(* IEC 61131-3 sources: verifaps-lib/share/PPU.stold (part 13) *)

(* ---- Scenario8_Final.xml.st ---- *)
TYPE
    Magazin_states_t : (Green_Lamp , Init , Interstep , Magazin_Init , Magazin_Init_2 , Slider_Move_Back , Start_Magazin , Step0 , Step1 , convey);
    Stamp_states_t : (Green_Lamp , Init , Interstep , Interstep_2 , StampProcess , StampSliderBack , StampSliderForward , Stamp_Init_1 , Stamp_Init_2 , Stamp_Init_3 , Stamp_Init_4 , Start_Stamp , Step0 , Step1 , Step2);
    Crane_states_t : (Crane_Go_Up , Crane_Go_Up_White , Crane_Init , Crane_Init_2 , Crane_Lift_At_Stamp , Crane_Lift_At_Stamp2 , Crane_Lift_Conveyor , Crane_Lift_Conveyor2 , Crane_Lift_Conveyor_Black , Crane_Lift_Magazin , Crane_Lift_Magazin_Metallic , Crane_Lift_Magazine_White , Crane_Lift_NOT_Metallic_Black , Crane_Lower , Crane_On_Conveyor , Crane_On_Conveyor_Metallic , Crane_On_Conveyor_Metallic2 , Crane_On_Conveyor_Not_Metallica_Black , Crane_On_Stamp_Metallic , Crane_On_Stamp_Metallic2 , Crane_On_Stamp_Metallic2_Lower , Crane_On_Stamp_Stop_Black , Crane_On_Stamp_White , Crane_Turn_Left_Back_To_Stamp , Crane_Turn_Left_From_Stamp , Crane_Turn_Left_Metallic , Crane_Turn_Left_Metallic2 , Crane_Turn_Left_NOT_Metallic , Crane_Turn_Left_NOT_Metallic_Black , Crane_Turn_Left_White , Crane_Turn_Right_From_Stamp , Init , Interstep , Interstep_2 , Interstep_3 , Interstep_4 , Lower_Crane , Magazin_Stop , Magazin_Stop_Black , Magazin_Stop_Final , No_Workpiece_ready , Reset_interconnect , Stamp_Pressure_Profile_Set_Metallic , Stamp_Pressure_Profile_Set_White , Start_Crane , Step0 , Step2 , Step3 , Step4 , Suck_At_Stamp , Suck_At_Stamp2 , TimeDelay , Turn_Right , Turn_Right_Black , Turn_Right_Final , pause , release , release2 , release_Black , release_Workpiece , release_Workpiece_White);
END_TYPE

FUNCTION_BLOCK Magazin
    VAR_INPUT  CraneDown : BOOL; END_VAR {*Irwxp*}
    VAR_OUTPUT  CraneLower : BOOL; END_VAR {*Orwxp*}
    VAR_INPUT  CraneOnConveyor : BOOL; END_VAR {*Irwxp*}
    VAR_INPUT  CraneOnMagazin : BOOL; END_VAR {*Irwxp*}
    VAR_INPUT  CraneSucked : BOOL; END_VAR {*Irwxp*}
    VAR_OUTPUT  CraneTurnClockwise : BOOL; END_VAR {*Orwxp*}
    VAR_OUTPUT  CraneTurnCounterclockwise : BOOL; END_VAR {*Orwxp*}
    VAR_INPUT  CraneUp : BOOL; END_VAR {*Irwxp*}
    VAR_OUTPUT  MagazinGreenLamp : BOOL; END_VAR {*Orwxp*}
    VAR_OUTPUT  MagazinSlider : BOOL; END_VAR {*Orwxp*}
    VAR_OUTPUT  MagazinVacuumOff : BOOL; END_VAR {*Orwxp*}
    VAR_OUTPUT  MagazinVacuumOn : BOOL; END_VAR {*Orwxp*}
    VAR_OUTPUT  MagazinWhiteLamp : BOOL; END_VAR {*Orwxp*}
    VAR  SFCInit : BOOL; END_VAR {*Lrwxp*}
    VAR_INPUT  SFCReset : BOOL; END_VAR {*Irwxp*}
    VAR_INPUT  SliderMovedOut : BOOL; END_VAR {*Irwxp*}
    VAR_INPUT  SliderNotMovedOut : BOOL; END_VAR {*Irwxp*}
    VAR_INPUT  StartButtonMagazin : BOOL; END_VAR {*Irwxp*}
    VAR_OUTPUT  StartCommandMagazin : BOOL; END_VAR {*Orwxp*}
    VAR_INPUT  StartVar : BOOL; END_VAR {*Irwxp*}
    VAR_INPUT  WorkpieceReady : BOOL; END_VAR {*Irwxp*}
    VAR  _state : Magazin_states_t; END_VAR {*Lrwxp*}
    VAR  _transit : BOOL; END_VAR {*Lrwxp*}
    VAR  interconnectMagazinStartCommand : BOOL; END_VAR {*Lrwxp*}

    CASE _state OF
        Magazin_states_t#Green_Lamp:
            _transit := FALSE;
            MagazinGreenLamp := TRUE;
            interconnectMagazinStartCommand := FALSE;
            IF TRUE THEN
                _transit := TRUE;
                _state := Magazin_states_t#Magazin_Init;
            END_IF;

        Magazin_states_t#Init:
            _transit := FALSE;
            IF TRUE THEN
                _transit := TRUE;
                _state := Magazin_states_t#Start_Magazin;
            END_IF;

        Magazin_states_t#Interstep:
            _transit := FALSE;
            StartCommandMagazin := TRUE;
            IF StartVar THEN
                _transit := TRUE;
                _state := Magazin_states_t#convey;
            END_IF;

        Magazin_states_t#Magazin_Init:
            _transit := FALSE;
            MagazinSlider := TRUE;
            IF TRUE THEN
                _transit := TRUE;
                _state := Magazin_states_t#Magazin_Init_2;
            END_IF;

        Magazin_states_t#Magazin_Init_2:
            _transit := FALSE;
            MagazinSlider := FALSE;
            IF TRUE THEN
                _transit := TRUE;
                _state := Magazin_states_t#Interstep;
            END_IF;

        Magazin_states_t#Slider_Move_Back:
            _transit := FALSE;
            IF ((SliderMovedOut = TRUE) AND (SliderNotMovedOut = FALSE)) THEN
                MagazinSlider := FALSE;
            END_IF;
            IF CraneUp THEN
                _transit := TRUE;
                _state := Magazin_states_t#Step1;
            END_IF;

        Magazin_states_t#Start_Magazin:
            _transit := FALSE;
            MagazinSlider := FALSE;
            MagazinGreenLamp := FALSE;
            StartVar := FALSE;
            StartCommandMagazin := FALSE;
            IF (StartButtonMagazin = TRUE) THEN
                interconnectMagazinStartCommand := TRUE;
            END_IF;
            IF interconnectMagazinStartCommand THEN
                _transit := TRUE;
                _state := Magazin_states_t#Green_Lamp;
            END_IF;

        Magazin_states_t#Step0:
            _transit := FALSE;
            IF CraneDown THEN
                _transit := TRUE;
                _state := Magazin_states_t#Slider_Move_Back;
            END_IF;

        Magazin_states_t#Step1:
            _transit := FALSE;
            IF CraneOnConveyor THEN
                _transit := TRUE;
                _state := Magazin_states_t#Interstep;
            END_IF;

        Magazin_states_t#convey:
            _transit := FALSE;
            IF SliderNotMovedOut THEN
                MagazinSlider := TRUE;
            END_IF;
            IF CraneOnMagazin THEN
                _transit := TRUE;
                _state := Magazin_states_t#Step0;
            END_IF;

            END_CASE;
END_FUNCTION_BLOCK

PROGRAM Main

VAR  Actuator_AnalogCranePressure : INT; END_VAR {*Lrwxp*}
VAR  Actuator_CraneLower : BOOL; END_VAR {*Lrwxp*}
VAR  Actuator_CraneTurnClockwise : BOOL; END_VAR {*Lrwxp*}
VAR  Actuator_CraneTurnCounterclockwise : BOOL; END_VAR {*Lrwxp*}
VAR  Actuator_MagazinGreenLamp : BOOL; END_VAR {*Lrwxp*}
VAR  Actuator_MagazinSlider : BOOL; END_VAR {*Lrwxp*}
VAR  Actuator_MagazinVacuumOff : BOOL; END_VAR {*Lrwxp*}
VAR  Actuator_MagazinVacuumOn : BOOL; END_VAR {*Lrwxp*}
VAR  Actuator_MagazinWhiteLamp : BOOL; END_VAR {*Lrwxp*}
VAR  Actuator_StampGreenLamp : BOOL; END_VAR {*Lrwxp*}
VAR  Actuator_StampPusher : BOOL; END_VAR {*Lrwxp*}
VAR  Actuator_StampSliderMovedIn : BOOL; END_VAR {*Lrwxp*}
VAR  Actuator_StampSliderMovedOut : BOOL; END_VAR {*Lrwxp*}
VAR  Actuator_StampWhiteLamp : BOOL; END_VAR {*Lrwxp*}
VAR  Crane : Crane; END_VAR {*Lrwxp*}
VAR  Mag : Magazin; END_VAR {*Lrwxp*}
VAR  Sensor_CraneDown : BOOL; END_VAR {*Lrwxp*}
VAR  Sensor_CraneOnConveyor : BOOL; END_VAR {*Lrwxp*}
VAR  Sensor_CraneOnMagazin : BOOL; END_VAR {*Lrwxp*}
VAR  Sensor_CranePosition : BOOL; END_VAR {*Lrwxp*}
VAR  Sensor_CranePositionStamp : BOOL; END_VAR {*Lrwxp*}
VAR  Sensor_CraneSucked : BOOL; END_VAR {*Lrwxp*}
VAR  Sensor_CraneUp : BOOL; END_VAR {*Lrwxp*}
VAR  Sensor_MagazinCapacitiveSensor : BOOL; END_VAR {*Lrwxp*}
VAR  Sensor_MagazinEmergencyStop : BOOL; END_VAR {*Lrwxp*}
VAR  Sensor_MagazinOpticalSensor : BOOL; END_VAR {*Lrwxp*}
VAR  Sensor_MagazinSwitchManuellAutomatic : BOOL; END_VAR {*Lrwxp*}
VAR  Sensor_SliderMovedOut : BOOL; END_VAR {*Lrwxp*}
VAR  Sensor_SliderNotMovedOut : BOOL; END_VAR {*Lrwxp*}
VAR  Sensor_StampEmergencyStop : BOOL; END_VAR {*Lrwxp*}
VAR  Sensor_StampLowered : BOOL; END_VAR {*Lrwxp*}
VAR  Sensor_StampSliderFilled : BOOL; END_VAR {*Lrwxp*}
VAR  Sensor_StampSliderSensorMovedIn : BOOL; END_VAR {*Lrwxp*}
VAR  Sensor_StampSliderSensorMovedOut : BOOL; END_VAR {*Lrwxp*}
VAR  Sensor_StampStartButton : BOOL; END_VAR {*Lrwxp*}
VAR  Sensor_StampSwitchManuellAutomatic : BOOL; END_VAR {*Lrwxp*}
VAR  Sensor_StampUp : BOOL; END_VAR {*Lrwxp*}
VAR  Sensor_StartButtonMagazin : BOOL; END_VAR {*Lrwxp*}
VAR  Sensor_WorkpieceReady : BOOL; END_VAR {*Lrwxp*}
VAR  Stamp : Stamp; END_VAR {*Lrwxp*}
Mag.SliderNotMovedOut := Sensor_SliderNotMovedOut;
Mag.SliderMovedOut := Sensor_SliderMovedOut;
Mag.CraneOnMagazin := Sensor_CraneOnMagazin;
Mag.CraneDown := Sensor_CraneDown;
Mag.CraneUp := Sensor_CraneUp;
Mag.CraneOnConveyor := Sensor_CraneOnConveyor;
Mag.WorkpieceReady := Sensor_WorkpieceReady;
Mag.StartButtonMagazin := Sensor_StartButtonMagazin;
Actuator_MagazinSlider := Mag.MagazinSlider;
Actuator_MagazinGreenLamp := Mag.MagazinGreenLamp;
Crane.CraneUp := Sensor_CraneUp;
Crane.CraneOnConveyor := Sensor_CraneOnConveyor;
Crane.CraneDown := Sensor_CraneDown;
Crane.CraneSucked := Sensor_CraneSucked;
Crane.CraneOnMagazin := Sensor_CraneOnMagazin;
Crane.MagazinCapacitiveSensor := Sensor_MagazinCapacitiveSensor;
Crane.CranePositionStamp := Sensor_CranePositionStamp;
Crane.SliderMovedOut := Sensor_SliderMovedOut;
Crane.WorkpieceReady := Sensor_WorkpieceReady;
Crane.MagazinOpticalSensor := Sensor_MagazinOpticalSensor;
Crane.StampSliderFilled := Sensor_StampSliderFilled;
Crane.StampSliderSensorMovedOut := Sensor_StampSliderSensorMovedOut;
Crane.StampLowered := Sensor_StampLowered;
Crane.StartButtonMagazin := Sensor_StartButtonMagazin;
Actuator_CraneTurnCounterclockwise := Crane.CraneTurnCounterclockwise;
Actuator_CraneTurnClockwise := Crane.CraneTurnClockwise;
Actuator_CraneLower := Crane.CraneLower;
Actuator_MagazinVacuumOff := Crane.MagazinVacuumOff;
Actuator_MagazinVacuumOn := Crane.MagazinVacuumOn;
Actuator_AnalogCranePressure := Crane.AnalogCranePressure;
Stamp.StampSliderSensorMovedOut := Sensor_StampSliderSensorMovedOut;
Stamp.StampSliderSensorMovedIn := Sensor_StampSliderSensorMovedIn;
Stamp.StampSliderFilled := Sensor_StampSliderFilled;
Stamp.StampUp := Sensor_StampUp;
Stamp.StampLowered := Sensor_StampLowered;
Stamp.CraneDown := Sensor_CraneDown;
Stamp.CraneUp := Sensor_CraneUp;
Stamp.CraneSucked := Sensor_CraneSucked;
Stamp.CranePositionStamp := Sensor_CranePositionStamp;
Stamp.CraneOnConveyor := Sensor_CraneOnConveyor;
Stamp.StampStartButton := Sensor_StampStartButton;
Actuator_StampSliderMovedOut := Stamp.StampSliderMovedOut;
Actuator_StampSliderMovedIn := Stamp.StampSliderMovedIn;
Actuator_StampWhiteLamp := Stamp.StampWhiteLamp;
Actuator_StampPusher := Stamp.StampPusher;
Actuator_StampGreenLamp := Stamp.StampGreenLamp;
IF (Sensor_StampEmergencyStop AND Sensor_MagazinEmergencyStop) THEN
    Mag();
    Crane();
    Stamp();
    IF (Actuator_MagazinGreenLamp AND Actuator_StampGreenLamp) THEN
        IF ((Stamp.StartCommandStamp AND Crane.StartCommandCrane) AND Mag.StartCommandMagazin) THEN
            Crane.StartVar := TRUE;
            Mag.StartVar := TRUE;
            Stamp.StartVar := TRUE;
        END_IF;
    END_IF;
    Crane.SFCReset := FALSE;
    Mag.SFCReset := FALSE;
    Stamp.SFCReset := FALSE;
ELSEIF (NOT Sensor_StampEmergencyStop OR NOT Sensor_MagazinEmergencyStop) THEN
    Actuator_MagazinSlider := FALSE;
    Actuator_CraneLower := FALSE;
    Actuator_MagazinVacuumOn := FALSE;
    Actuator_MagazinVacuumOff := TRUE;
    Actuator_MagazinGreenLamp := FALSE;
    Actuator_CraneTurnCounterclockwise := FALSE;
    Actuator_CraneTurnClockwise := FALSE;
    Actuator_StampSliderMovedOut := TRUE;
    Actuator_StampSliderMovedIn := FALSE;
    Actuator_StampGreenLamp := FALSE;
    Actuator_StampPusher := FALSE;
    Actuator_AnalogCranePressure := INT#0;
    Crane.SFCReset := TRUE;
    Mag.SFCReset := TRUE;
    Stamp.SFCReset := TRUE;
    Crane.StartVar := FALSE;
    Mag.StartVar := FALSE;
    Stamp.StartVar := FALSE;
END_IF;
END_PROGRAM
FUNCTION_BLOCK Stamp
VAR_INPUT  CraneDown : BOOL; END_VAR {*Irwxp*}
VAR_INPUT  CraneOnConveyor : BOOL; END_VAR {*Irwxp*}
VAR_INPUT  CranePositionStamp : BOOL; END_VAR {*Irwxp*}
VAR_INPUT  CraneSucked : BOOL; END_VAR {*Irwxp*}
VAR_INPUT  CraneUp : BOOL; END_VAR {*Irwxp*}
VAR  Duration : TIME := TIME#500.0ms; END_VAR {*Lrwxp*}
VAR  SFCInit : BOOL; END_VAR {*Lrwxp*}
VAR_INPUT  SFCReset : BOOL; END_VAR {*Irwxp*}
VAR_OUTPUT  StampGreenLamp : BOOL; END_VAR {*Orwxp*}
VAR_INPUT  StampLowered : BOOL; END_VAR {*Irwxp*}
VAR_OUTPUT  StampPressure : BOOL; END_VAR {*Orwxp*}
VAR_OUTPUT  StampPusher : BOOL; END_VAR {*Orwxp*}
VAR_INPUT  StampSliderFilled : BOOL; END_VAR {*Irwxp*}
VAR_OUTPUT  StampSliderMovedIn : BOOL; END_VAR {*Orwxp*}
VAR_OUTPUT  StampSliderMovedOut : BOOL; END_VAR {*Orwxp*}
VAR_INPUT  StampSliderSensorMovedIn : BOOL; END_VAR {*Irwxp*}
VAR_INPUT  StampSliderSensorMovedOut : BOOL; END_VAR {*Irwxp*}
VAR_INPUT  StampStartButton : BOOL; END_VAR {*Irwxp*}
VAR_INPUT  StampUp : BOOL; END_VAR {*Irwxp*}
VAR_OUTPUT  StampWhiteLamp : BOOL; END_VAR {*Orwxp*}
VAR_OUTPUT  StartCommandStamp : BOOL; END_VAR {*Orwxp*}
VAR_INPUT  StartVar : BOOL; END_VAR {*Irwxp*}
VAR  Timer : TON; END_VAR {*Lrwxp*}
VAR  _state : Stamp_states_t; END_VAR {*Lrwxp*}
VAR  _transit : BOOL; END_VAR {*Lrwxp*}
VAR  interconnect : BOOL; END_VAR {*Lrwxp*}
VAR  interconnectStampStartCommand : BOOL; END_VAR {*Lrwxp*}

CASE _state OF
    Stamp_states_t#Green_Lamp:
        _transit := FALSE;
        StampGreenLamp := TRUE;
        interconnectStampStartCommand := FALSE;
        IF TRUE THEN
            _transit := TRUE;
            _state := Stamp_states_t#Stamp_Init_1;
        END_IF;

    Stamp_states_t#Init:
        _transit := FALSE;
        IF TRUE THEN
            _transit := TRUE;
            _state := Stamp_states_t#Start_Stamp;
        END_IF;

    Stamp_states_t#Interstep:
        _transit := FALSE;
        StartCommandStamp := TRUE;
        IF StartVar THEN
            _transit := TRUE;
            _state := Stamp_states_t#Interstep_2;
        END_IF;

    Stamp_states_t#Interstep_2:
        _transit := FALSE;
        IF StampSliderFilled THEN
            _transit := TRUE;
            _state := Stamp_states_t#Step0;
        END_IF;

    Stamp_states_t#StampProcess:
        _transit := FALSE;
        StampSliderMovedIn := FALSE;
        StampPusher := TRUE;
        IF StampLowered THEN
            _transit := TRUE;
            _state := Stamp_states_t#Step1;
        END_IF;

    Stamp_states_t#StampSliderBack:
        _transit := FALSE;
        StampSliderMovedIn := TRUE;
        StampSliderMovedOut := FALSE;
        IF StampSliderSensorMovedIn THEN
            _transit := TRUE;
            _state := Stamp_states_t#StampProcess;
        END_IF;

    Stamp_states_t#StampSliderForward:
        _transit := FALSE;
        StampPusher := FALSE;
        StampSliderMovedOut := TRUE;
        IF ((StampLowered = FALSE) AND (StampUp = TRUE)) THEN
            interconnect := FALSE;
        END_IF;
        Timer(IN := FALSE, PT := TIME#1.0ms);
        IF StampSliderMovedOut THEN
            _transit := TRUE;
            _state := Stamp_states_t#Step2;
        END_IF;

    Stamp_states_t#Stamp_Init_1:
        _transit := FALSE;
        StampSliderMovedIn := TRUE;
        StampSliderMovedOut := FALSE;
        IF StampSliderSensorMovedIn THEN
            _transit := TRUE;
            _state := Stamp_states_t#Stamp_Init_2;
        END_IF;

    Stamp_states_t#Stamp_Init_2:
        _transit := FALSE;
        StampSliderMovedIn := FALSE;
        StampSliderMovedOut := TRUE;
        IF StampSliderSensorMovedOut THEN
            _transit := TRUE;
            _state := Stamp_states_t#Stamp_Init_3;
        END_IF;

    Stamp_states_t#Stamp_Init_3:
        _transit := FALSE;
        StampPusher := TRUE;
        IF StampLowered THEN
            _transit := TRUE;
            _state := Stamp_states_t#Stamp_Init_4;
        END_IF;

    Stamp_states_t#Stamp_Init_4:
        _transit := FALSE;
        StampPusher := FALSE;
        IF StampUp THEN
            _transit := TRUE;
            _state := Stamp_states_t#Interstep;
        END_IF;

    Stamp_states_t#Start_Stamp:
        _transit := FALSE;
        StampSliderMovedOut := FALSE;
        StampSliderMovedIn := FALSE;
        StampPusher := FALSE;
        StampGreenLamp := FALSE;
        StampPressure := FALSE;
        StartCommandStamp := FALSE;
        IF (StampStartButton = TRUE) THEN
            interconnectStampStartCommand := TRUE;
        END_IF;
        IF interconnectStampStartCommand THEN
            _transit := TRUE;
            _state := Stamp_states_t#Green_Lamp;
        END_IF;

    Stamp_states_t#Step0:
        _transit := FALSE;
        IF CraneUp THEN
            _transit := TRUE;
            _state := Stamp_states_t#StampSliderBack;
        END_IF;

    Stamp_states_t#Step1:
        _transit := FALSE;
        Timer(IN := StampLowered, PT := TIME#);
        interconnect := Timer.Q;
        IF interconnect THEN
            _transit := TRUE;
            _state := Stamp_states_t#StampSliderForward;
        END_IF;

    Stamp_states_t#Step2:
        _transit := FALSE;
        IF (CraneOnConveyor AND NOT StampSliderFilled) THEN
            _transit := TRUE;
            _state := Stamp_states_t#Interstep;
        END_IF;

    END_CASE;
END_FUNCTION_BLOCK

FUNCTION_BLOCK Crane
VAR_OUTPUT  AnalogCranePressure : INT; END_VAR {*Orwxp*}
VAR_INPUT  CraneDown : BOOL; END_VAR {*Irwxp*}
VAR_OUTPUT  CraneLower : BOOL; END_VAR {*Orwxp*}
VAR_INPUT  CraneOnConveyor : BOOL; END_VAR {*Irwxp*}
VAR_INPUT  CraneOnMagazin : BOOL; END_VAR {*Irwxp*}
VAR_INPUT  CranePositionStamp : BOOL; END_VAR {*Irwxp*}
VAR_INPUT  CraneSucked : BOOL; END_VAR {*Irwxp*}
VAR_OUTPUT  CraneTurnClockwise : BOOL; END_VAR {*Orwxp*}
VAR_OUTPUT  CraneTurnCounterclockwise : BOOL; END_VAR {*Orwxp*}
VAR_INPUT  CraneUp : BOOL; END_VAR {*Irwxp*}
VAR  Duration1 : TIME := TIME#1.0s500.0ms; END_VAR {*Lrwxp*}
VAR_INPUT  MagazinCapacitiveSensor : BOOL; END_VAR {*Irwxp*}
VAR_INPUT  MagazinOpticalSensor : BOOL; END_VAR {*Irwxp*}
VAR_OUTPUT  MagazinVacuumOff : BOOL; END_VAR {*Orwxp*}
VAR_OUTPUT  MagazinVacuumOn : BOOL; END_VAR {*Orwxp*}
VAR  SFCInit : BOOL; END_VAR {*Lrwxp*}
VAR_INPUT  SFCReset : BOOL; END_VAR {*Irwxp*}
VAR_INPUT  SliderMovedOut : BOOL; END_VAR {*Irwxp*}
VAR_INPUT  SliderNotMovedOut : BOOL; END_VAR {*Irwxp*}
VAR_INPUT  StampLowered : BOOL; END_VAR {*Irwxp*}
VAR_INPUT  StampSliderFilled : BOOL; END_VAR {*Irwxp*}
VAR_INPUT  StampSliderSensorMovedOut : BOOL; END_VAR {*Irwxp*}
VAR_INPUT  StartButtonMagazin : BOOL; END_VAR {*Irwxp*}
VAR_OUTPUT  StartCommandCrane : BOOL; END_VAR {*Orwxp*}
VAR_INPUT  StartVar : BOOL; END_VAR {*Irwxp*}
VAR  TimeDelay_Timer : TON; END_VAR {*Lrwxp*}
VAR  TimeDelay_Timer_Duration : TIME := TIME#50.0ms; END_VAR {*Lrwxp*}
VAR  TimeDelay_Timer_interconnect : BOOL; END_VAR {*Lrwxp*}
VAR  Timer1 : TON; END_VAR {*Lrwxp*}
VAR_INPUT  WorkpieceReady : BOOL; END_VAR {*Irwxp*}
VAR  _state : Crane_states_t; END_VAR {*Lrwxp*}
VAR  _transit : BOOL; END_VAR {*Lrwxp*}
VAR  actualtime1 : TIME; END_VAR {*Lrwxp*}
VAR  interconnect : BOOL; END_VAR {*Lrwxp*}
VAR  interconnectCraneStartCommand : BOOL; END_VAR {*Lrwxp*}

CASE _state OF
    Crane_states_t#Crane_Go_Up:
        _transit := FALSE;
        CraneLower := FALSE;
        IF CraneUp THEN
            _transit := TRUE;
            _state := Crane_states_t#Step3;
        END_IF;

    Crane_states_t#Crane_Go_Up_White:
        _transit := FALSE;
        CraneLower := FALSE;
        IF CraneUp THEN
            _transit := TRUE;
            _state := Crane_states_t#Step3;
        END_IF;

    Crane_states_t#Crane_Init:
        _transit := FALSE;
        CraneLower := TRUE;
        interconnectCraneStartCommand := FALSE;
        AnalogCranePressure := INT#6000;
        IF CraneDown THEN
            _transit := TRUE;
            _state := Crane_states_t#Crane_Init_2;
        END_IF;

    Crane_states_t#Crane_Init_2:
        _transit := FALSE;
        CraneLower := FALSE;
        IF CraneUp THEN
            _transit := TRUE;
            _state := Crane_states_t#Interstep;
        END_IF;

    Crane_states_t#Crane_Lift_At_Stamp:
        _transit := FALSE;
        CraneLower := FALSE;
        IF CraneUp THEN
            _transit := TRUE;
            _state := Crane_states_t#Crane_Turn_Left_From_Stamp;
        END_IF;

    Crane_states_t#Crane_Lift_At_Stamp2:
        _transit := FALSE;
        CraneLower := FALSE;
        IF CraneUp THEN
            _transit := TRUE;
            _state := Crane_states_t#Crane_Turn_Right_From_Stamp;
        END_IF;

    Crane_states_t#Crane_Lift_Conveyor:
        _transit := FALSE;
        CraneLower := FALSE;
        IF TRUE THEN
            _transit := TRUE;
            _state := Crane_states_t#Interstep;
        END_IF;

    Crane_states_t#Crane_Lift_Conveyor2:
        _transit := FALSE;
        CraneLower := FALSE;
        IF TRUE THEN
            _transit := TRUE;
            _state := Crane_states_t#Interstep;
        END_IF;

    Crane_states_t#Crane_Lift_Conveyor_Black:
        _transit := FALSE;
        CraneLower := FALSE;
        IF CraneUp THEN
            _transit := TRUE;
            _state := Crane_states_t#Crane_Turn_Left_Back_To_Stamp;
        END_IF;

    Crane_states_t#Crane_Lift_Magazin:
        _transit := FALSE;
        CraneLower := FALSE;
        IF CraneUp THEN
            _transit := TRUE;
            _state := Crane_states_t#Crane_Turn_Left_NOT_Metallic;
        END_IF;

    Crane_states_t#Crane_Lift_Magazin_Metallic:
        _transit := FALSE;
        CraneLower := FALSE;
        IF CraneUp THEN
            _transit := TRUE;
            _state := Crane_states_t#Crane_Turn_Left_Metallic;
        END_IF;

    Crane_states_t#Crane_Lift_Magazine_White:
        _transit := FALSE;
        CraneLower := FALSE;
        IF CraneUp THEN
            _transit := TRUE;
            _state := Crane_states_t#Crane_Turn_Left_White;
        END_IF;

    Crane_states_t#Crane_Lift_NOT_Metallic_Black:
        _transit := FALSE;
        CraneLower := FALSE;
        IF CraneUp THEN
            _transit := TRUE;
            _state := Crane_states_t#Crane_Turn_Left_NOT_Metallic_Black;
        END_IF;

    Crane_states_t#Crane_Lower:
        _transit := FALSE;
        MagazinVacuumOn := TRUE;
        MagazinVacuumOff := FALSE;
        CraneLower := TRUE;
        AnalogCranePressure := INT#0;
        IF CraneSucked THEN
            _transit := TRUE;
            _state := Crane_states_t#Step0;
        END_IF;

    Crane_states_t#Crane_On_Conveyor:
        _transit := FALSE;
        CraneTurnCounterclockwise := FALSE;
        CraneTurnClockwise := FALSE;
        CraneLower := TRUE;
        IF CraneDown THEN
            _transit := TRUE;
            _state := Crane_states_t#release;
        END_IF;

    Crane_states_t#Crane_On_Conveyor_Metallic:
        _transit := FALSE;
        CraneTurnCounterclockwise := FALSE;
        CraneTurnClockwise := FALSE;
        CraneLower := TRUE;
        IF CraneDown THEN
            _transit := TRUE;
            _state := Crane_states_t#release;
        END_IF;

    Crane_states_t#Crane_On_Conveyor_Metallic2:
        _transit := FALSE;
        CraneTurnCounterclockwise := FALSE;
        CraneTurnClockwise := FALSE;
        CraneLower := TRUE;
        IF CraneDown THEN
            _transit := TRUE;
            _state := Crane_states_t#release2;
        END_IF;

    Crane_states_t#Crane_On_Conveyor_Not_Metallica_Black:
        _transit := FALSE;
        CraneTurnCounterclockwise := FALSE;
        CraneTurnClockwise := FALSE;
        CraneLower := TRUE;
        IF CraneDown THEN
            _transit := TRUE;
            _state := Crane_states_t#release_Black;
        END_IF;

    Crane_states_t#Crane_On_Stamp_Metallic:
        _transit := FALSE;
        CraneTurnCounterclockwise := FALSE;
        CraneTurnClockwise := FALSE;
        CraneLower := TRUE;
        IF CraneDown THEN
            _transit := TRUE;
            _state := Crane_states_t#release_Workpiece;
        END_IF;

    Crane_states_t#Crane_On_Stamp_Metallic2:
        _transit := FALSE;
        CraneTurnCounterclockwise := FALSE;
        CraneTurnClockwise := FALSE;
        IF StampLowered THEN
            _transit := TRUE;
            _state := Crane_states_t#Interstep_4;
        END_IF;

    Crane_states_t#Crane_On_Stamp_Metallic2_Lower:
        _transit := FALSE;
        CraneLower := TRUE;
        IF CraneDown THEN
            _transit := TRUE;
            _state := Crane_states_t#Suck_At_Stamp2;
        END_IF;

    Crane_states_t#Crane_On_Stamp_Stop_Black:
        _transit := FALSE;
        CraneTurnClockwise := FALSE;
        CraneTurnCounterclockwise := FALSE;
        IF TRUE THEN
            _transit := TRUE;
            _state := Crane_states_t#Reset_interconnect;
        END_IF;

    Crane_states_t#Crane_On_Stamp_White:
        _transit := FALSE;
        CraneTurnCounterclockwise := FALSE;
        CraneTurnClockwise := FALSE;
        CraneLower := TRUE;
        IF CraneDown THEN
            _transit := TRUE;
            _state := Crane_states_t#release_Workpiece_White;
        END_IF;

    Crane_states_t#Crane_Turn_Left_Back_To_Stamp:
        _transit := FALSE;
        CraneTurnCounterclockwise := TRUE;
        CraneTurnClockwise := FALSE;
        IF CranePositionStamp THEN
            _transit := TRUE;
            _state := Crane_states_t#Crane_On_Stamp_Stop_Black;
        END_IF;

    Crane_states_t#Crane_Turn_Left_From_Stamp:
        _transit := FALSE;
        CraneTurnClockwise := TRUE;
        CraneTurnCounterclockwise := FALSE;
        IF CraneOnConveyor THEN
            _transit := TRUE;
            _state := Crane_states_t#Crane_On_Conveyor_Metallic;
        END_IF;

    Crane_states_t#Crane_Turn_Left_Metallic:
        _transit := FALSE;
        CraneTurnCounterclockwise := TRUE;
        CraneTurnClockwise := FALSE;
        IF CranePositionStamp THEN
            _transit := TRUE;
            _state := Crane_states_t#Crane_On_Stamp_Metallic;
        END_IF;

    Crane_states_t#Crane_Turn_Left_Metallic2:
        _transit := FALSE;
        CraneTurnCounterclockwise := TRUE;
        CraneTurnClockwise := FALSE;
        IF CranePositionStamp THEN
            _transit := TRUE;
            _state := Crane_states_t#Crane_On_Stamp_Metallic2;
        END_IF;

    Crane_states_t#Crane_Turn_Left_NOT_Metallic:
        _transit := FALSE;
        CraneTurnCounterclockwise := TRUE;
        CraneTurnClockwise := FALSE;
        IF CraneOnConveyor THEN
            _transit := TRUE;
            _state := Crane_states_t#Crane_On_Conveyor;
        END_IF;

    Crane_states_t#Crane_Turn_Left_NOT_Metallic_Black:
        _transit := FALSE;
        CraneTurnCounterclockwise := TRUE;
        CraneTurnClockwise := FALSE;
        IF CraneOnConveyor THEN
            _transit := TRUE;
            _state := Crane_states_t#Crane_On_Conveyor_Not_Metallica_Black;
        END_IF;

    Crane_states_t#Crane_Turn_Left_White:
        _transit := FALSE;
        CraneTurnCounterclockwise := TRUE;
        CraneTurnClockwise := FALSE;
        IF CranePositionStamp THEN
            _transit := TRUE;
            _state := Crane_states_t#Crane_On_Stamp_White;
        END_IF;

    Crane_states_t#Crane_Turn_Right_From_Stamp:
        _transit := FALSE;
        CraneTurnClockwise := TRUE;
        CraneTurnCounterclockwise := FALSE;
        IF CraneOnConveyor THEN
            _transit := TRUE;
            _state := Crane_states_t#Crane_On_Conveyor_Metallic2;
        END_IF;

    Crane_states_t#Init:
        _transit := FALSE;
        IF TRUE THEN
            _transit := TRUE;
            _state := Crane_states_t#Start_Crane;
        END_IF;

    Crane_states_t#Interstep:
        _transit := FALSE;
        StartCommandCrane := TRUE;
        IF StartVar THEN
            _transit := TRUE;
            _state := Crane_states_t#Interstep_2;
        END_IF;

    Crane_states_t#Interstep_2:
        _transit := FALSE;
        IF SliderMovedOut THEN
            _transit := TRUE;
            _state := Crane_states_t#TimeDelay;
        END_IF;

    Crane_states_t#Interstep_3:
        _transit := FALSE;
        IF NOT WorkpieceReady THEN
            _transit := TRUE;
            _state := Crane_states_t#No_Workpiece_ready;
        ELSEIF WorkpieceReady THEN
            _transit := TRUE;
            _state := Crane_states_t#Turn_Right;
        END_IF;

    Crane_states_t#Interstep_4:
        _transit := FALSE;
        IF StampSliderSensorMovedOut THEN
            _transit := TRUE;
            _state := Crane_states_t#Crane_On_Stamp_Metallic2_Lower;
        END_IF;

    Crane_states_t#Lower_Crane:
        _transit := FALSE;
        CraneLower := TRUE;
        IF CraneDown THEN
            _transit := TRUE;
            _state := Crane_states_t#Suck_At_Stamp;
        END_IF;

    Crane_states_t#Magazin_Stop:
        _transit := FALSE;
        CraneTurnClockwise := FALSE;
        CraneTurnCounterclockwise := FALSE;
        IF TRUE THEN
            _transit := TRUE;
            _state := Crane_states_t#Crane_Lower;
        END_IF;

    Crane_states_t#Magazin_Stop_Black:
        _transit := FALSE;
        CraneTurnClockwise := FALSE;
        CraneTurnCounterclockwise := FALSE;
        MagazinVacuumOn := TRUE;
        MagazinVacuumOff := FALSE;
        CraneLower := TRUE;
        IF CraneSucked THEN
            _transit := TRUE;
            _state := Crane_states_t#Crane_Lift_NOT_Metallic_Black;
        END_IF;

    Crane_states_t#Magazin_Stop_Final:
        _transit := FALSE;
        CraneTurnClockwise := FALSE;
        CraneTurnCounterclockwise := FALSE;
        IF TRUE THEN
            _transit := TRUE;
            _state := Crane_states_t#Start_Crane;
        END_IF;

    Crane_states_t#No_Workpiece_ready:
        _transit := FALSE;
        MagazinVacuumOn := FALSE;
        MagazinVacuumOff := FALSE;
        CraneLower := FALSE;
        IF NOT StampSliderFilled THEN
            _transit := TRUE;
            _state := Crane_states_t#Turn_Right_Final;
        ELSEIF StampSliderFilled THEN
            _transit := TRUE;
            _state := Crane_states_t#Crane_Turn_Left_Metallic2;
        END_IF;

    Crane_states_t#Reset_interconnect:
        _transit := FALSE;
        interconnect := FALSE;
        Timer1(IN := FALSE, PT := TIME#1.0ms);
        IF SliderMovedOut THEN
            _transit := TRUE;
            _state := Crane_states_t#Lower_Crane;
        END_IF;

    Crane_states_t#Stamp_Pressure_Profile_Set_Metallic:
        _transit := FALSE;
        AnalogCranePressure := INT#7000;
        IF TRUE THEN
            _transit := TRUE;
            _state := Crane_states_t#Crane_Lift_Magazin_Metallic;
        END_IF;

    Crane_states_t#Stamp_Pressure_Profile_Set_White:
        _transit := FALSE;
        AnalogCranePressure := INT#6000;
        IF TRUE THEN
            _transit := TRUE;
            _state := Crane_states_t#Crane_Lift_Magazine_White;
        END_IF;

    Crane_states_t#Start_Crane:
        _transit := FALSE;
        CraneLower := FALSE;
        MagazinVacuumOff := TRUE;
        MagazinVacuumOn := FALSE;
        CraneTurnCounterclockwise := FALSE;
        CraneTurnClockwise := FALSE;
        StartVar := FALSE;
        StartCommandCrane := FALSE;
        IF (StartButtonMagazin = TRUE) THEN
            interconnectCraneStartCommand := TRUE;
        END_IF;
        IF interconnectCraneStartCommand THEN
            _transit := TRUE;
            _state := Crane_states_t#Crane_Init;
        END_IF;

    Crane_states_t#Step0:
        _transit := FALSE;
        IF (NOT MagazinCapacitiveSensor AND MagazinOpticalSensor) THEN
            _transit := TRUE;
            _state := Crane_states_t#Stamp_Pressure_Profile_Set_White;
        ELSEIF (MagazinCapacitiveSensor AND MagazinOpticalSensor) THEN
            _transit := TRUE;
            _state := Crane_states_t#Stamp_Pressure_Profile_Set_Metallic;
        ELSEIF (NOT MagazinCapacitiveSensor AND NOT MagazinOpticalSensor) THEN
            _transit := TRUE;
            _state := Crane_states_t#Crane_Lift_Magazin;
        END_IF;

    Crane_states_t#Step2:
        _transit := FALSE;
        IF (MagazinCapacitiveSensor OR MagazinOpticalSensor) THEN
            _transit := TRUE;
            _state := Crane_states_t#pause;
        ELSEIF (NOT MagazinCapacitiveSensor AND NOT MagazinOpticalSensor) THEN
            _transit := TRUE;
            _state := Crane_states_t#Turn_Right_Black;
        END_IF;

    Crane_states_t#Step3:
        _transit := FALSE;
        IF NOT WorkpieceReady THEN
            _transit := TRUE;
            _state := Crane_states_t#Step4;
        ELSEIF WorkpieceReady THEN
            _transit := TRUE;
            _state := Crane_states_t#Step2;
        END_IF;

    Crane_states_t#Step4:
        _transit := FALSE;
        IF TRUE THEN
            _transit := TRUE;
            _state := Crane_states_t#Interstep;
        END_IF;

    Crane_states_t#Suck_At_Stamp:
        _transit := FALSE;
        MagazinVacuumOn := TRUE;
        MagazinVacuumOff := FALSE;
        IF CraneSucked THEN
            _transit := TRUE;
            _state := Crane_states_t#Crane_Lift_At_Stamp;
        END_IF;

    Crane_states_t#Suck_At_Stamp2:
        _transit := FALSE;
        MagazinVacuumOn := TRUE;
        MagazinVacuumOff := FALSE;
        IF CraneSucked THEN
            _transit := TRUE;
            _state := Crane_states_t#Crane_Lift_At_Stamp2;
        END_IF;

    Crane_states_t#TimeDelay:
        _transit := FALSE;
        TimeDelay_Timer(IN := TRUE, PT := TimeDelay_Timer_Duration);
        TimeDelay_Timer_interconnect := TimeDelay_Timer.Q;
        IF TimeDelay_Timer_interconnect THEN
            _transit := TRUE;
            _state := Crane_states_t#Interstep_3;
        END_IF;

    Crane_states_t#Turn_Right:
        _transit := FALSE;
        CraneTurnClockwise := TRUE;
        CraneTurnCounterclockwise := FALSE;
        IF CraneOnMagazin THEN
            _transit := TRUE;
            _state := Crane_states_t#Magazin_Stop;
        END_IF;

    Crane_states_t#Turn_Right_Black:
        _transit := FALSE;
        CraneTurnClockwise := TRUE;
        CraneTurnCounterclockwise := FALSE;
        IF CraneOnMagazin THEN
            _transit := TRUE;
            _state := Crane_states_t#Magazin_Stop_Black;
        END_IF;

    Crane_states_t#Turn_Right_Final:
        _transit := FALSE;
        CraneTurnClockwise := TRUE;
        CraneTurnCounterclockwise := FALSE;
        AnalogCranePressure := INT#0;
        IF CraneOnMagazin THEN
            _transit := TRUE;
            _state := Crane_states_t#Magazin_Stop_Final;
        END_IF;

    Crane_states_t#pause:
        _transit := FALSE;
        Timer1(IN := CraneUp, PT := Duration1);
        interconnect := Timer1.Q;
        IF interconnect THEN
            _transit := TRUE;
            _state := Crane_states_t#Reset_interconnect;
        END_IF;

    Crane_states_t#release:
        _transit := FALSE;
        MagazinVacuumOff := TRUE;
        MagazinVacuumOn := FALSE;
        IF TRUE THEN
            _transit := TRUE;
            _state := Crane_states_t#Crane_Lift_Conveyor;
        END_IF;

    Crane_states_t#release2:
        _transit := FALSE;
        MagazinVacuumOff := TRUE;
        MagazinVacuumOn := FALSE;
        IF TRUE THEN
            _transit := TRUE;
            _state := Crane_states_t#Crane_Lift_Conveyor2;
        END_IF;

    Crane_states_t#release_Black:
        _transit := FALSE;
        MagazinVacuumOn := FALSE;
        MagazinVacuumOff := TRUE;
        IF TRUE THEN
            _transit := TRUE;
            _state := Crane_states_t#Crane_Lift_Conveyor_Black;
        END_IF;

    Crane_states_t#release_Workpiece:
        _transit := FALSE;
        MagazinVacuumOff := TRUE;
        MagazinVacuumOn := FALSE;
        IF TRUE THEN
            _transit := TRUE;
            _state := Crane_states_t#Crane_Go_Up;
        END_IF;

    Crane_states_t#release_Workpiece_White:
        _transit := FALSE;
        MagazinVacuumOff := TRUE;
        MagazinVacuumOn := FALSE;
        IF TRUE THEN
            _transit := TRUE;
            _state := Crane_states_t#Crane_Go_Up_White;
        END_IF;

    END_CASE;
END_FUNCTION_BLOCK

(* ---- Scenario8_Final.xml_Crane.st ---- *)
FUNCTION_BLOCK Crane
    VAR_OUTPUT  AnalogCranePressure : INT; END_VAR {*Orwxp*}
    VAR_INPUT  CraneDown : BOOL; END_VAR {*Irwxp*}
    VAR_OUTPUT  CraneLower : BOOL; END_VAR {*Orwxp*}
    VAR_INPUT  CraneOnConveyor : BOOL; END_VAR {*Irwxp*}
    VAR_INPUT  CraneOnMagazin : BOOL; END_VAR {*Irwxp*}
    VAR_INPUT  CranePositionStamp : BOOL; END_VAR {*Irwxp*}
    VAR_INPUT  CraneSucked : BOOL; END_VAR {*Irwxp*}
    VAR_OUTPUT  CraneTurnClockwise : BOOL; END_VAR {*Orwxp*}
    VAR_OUTPUT  CraneTurnCounterclockwise : BOOL; END_VAR {*Orwxp*}
    VAR_INPUT  CraneUp : BOOL; END_VAR {*Irwxp*}
    VAR  Duration1 : TIME := TIME#1.0s500.0ms; END_VAR {*Lrwxp*}
    VAR_INPUT  MagazinCapacitiveSensor : BOOL; END_VAR {*Irwxp*}
    VAR_INPUT  MagazinOpticalSensor : BOOL; END_VAR {*Irwxp*}
    VAR_OUTPUT  MagazinVacuumOff : BOOL; END_VAR {*Orwxp*}
    VAR_OUTPUT  MagazinVacuumOn : BOOL; END_VAR {*Orwxp*}
    VAR  SFCInit : BOOL; END_VAR {*Lrwxp*}
    VAR_INPUT  SFCReset : BOOL; END_VAR {*Irwxp*}
    VAR_INPUT  SliderMovedOut : BOOL; END_VAR {*Irwxp*}
    VAR_INPUT  SliderNotMovedOut : BOOL; END_VAR {*Irwxp*}
    VAR_INPUT  StampLowered : BOOL; END_VAR {*Irwxp*}
    VAR_INPUT  StampSliderFilled : BOOL; END_VAR {*Irwxp*}
    VAR_INPUT  StampSliderSensorMovedOut : BOOL; END_VAR {*Irwxp*}
    VAR_INPUT  StartButtonMagazin : BOOL; END_VAR {*Irwxp*}
    VAR_OUTPUT  StartCommandCrane : BOOL; END_VAR {*Orwxp*}
    VAR_INPUT  StartVar : BOOL; END_VAR {*Irwxp*}
    VAR  TimeDelay_Timer : TON; END_VAR {*Lrwxp*}
    VAR  TimeDelay_Timer_Duration : TIME := TIME#50.0ms; END_VAR {*Lrwxp*}
    VAR  TimeDelay_Timer_interconnect : BOOL; END_VAR {*Lrwxp*}
    VAR  Timer1 : TON; END_VAR {*Lrwxp*}
    VAR_INPUT  WorkpieceReady : BOOL; END_VAR {*Irwxp*}
    VAR  _state : Crane_states_t; END_VAR {*Lrwxp*}
    VAR  _transit : BOOL; END_VAR {*Lrwxp*}
    VAR  actualtime1 : TIME; END_VAR {*Lrwxp*}
    VAR  interconnect : BOOL; END_VAR {*Lrwxp*}
    VAR  interconnectCraneStartCommand : BOOL; END_VAR {*Lrwxp*}

    CASE _state OF
        Crane_states_t#Crane_Go_Up:
            _transit := FALSE;
            CraneLower := FALSE;
            IF CraneUp THEN
                _transit := TRUE;
                _state := Crane_states_t#Step3;
            END_IF;

        Crane_states_t#Crane_Go_Up_White:
            _transit := FALSE;
            CraneLower := FALSE;
            IF CraneUp THEN
                _transit := TRUE;
                _state := Crane_states_t#Step3;
            END_IF;

        Crane_states_t#Crane_Init:
            _transit := FALSE;
            CraneLower := TRUE;
            interconnectCraneStartCommand := FALSE;
            AnalogCranePressure := INT#6000;
            IF CraneDown THEN
                _transit := TRUE;
                _state := Crane_states_t#Crane_Init_2;
            END_IF;

        Crane_states_t#Crane_Init_2:
            _transit := FALSE;
            CraneLower := FALSE;
            IF CraneUp THEN
                _transit := TRUE;
                _state := Crane_states_t#Interstep;
            END_IF;

        Crane_states_t#Crane_Lift_At_Stamp:
            _transit := FALSE;
            CraneLower := FALSE;
            IF CraneUp THEN
                _transit := TRUE;
                _state := Crane_states_t#Crane_Turn_Left_From_Stamp;
            END_IF;

        Crane_states_t#Crane_Lift_At_Stamp2:
            _transit := FALSE;
            CraneLower := FALSE;
            IF CraneUp THEN
                _transit := TRUE;
                _state := Crane_states_t#Crane_Turn_Right_From_Stamp;
            END_IF;

        Crane_states_t#Crane_Lift_Conveyor:
            _transit := FALSE;
            CraneLower := FALSE;
            IF TRUE THEN
                _transit := TRUE;
                _state := Crane_states_t#Interstep;
            END_IF;

        Crane_states_t#Crane_Lift_Conveyor2:
            _transit := FALSE;
            CraneLower := FALSE;
            IF TRUE THEN
                _transit := TRUE;
                _state := Crane_states_t#Interstep;
            END_IF;

        Crane_states_t#Crane_Lift_Conveyor_Black:
            _transit := FALSE;
            CraneLower := FALSE;
            IF CraneUp THEN
                _transit := TRUE;
                _state := Crane_states_t#Crane_Turn_Left_Back_To_Stamp;
            END_IF;

        Crane_states_t#Crane_Lift_Magazin:
            _transit := FALSE;
            CraneLower := FALSE;
            IF CraneUp THEN
                _transit := TRUE;
                _state := Crane_states_t#Crane_Turn_Left_NOT_Metallic;
            END_IF;

        Crane_states_t#Crane_Lift_Magazin_Metallic:
            _transit := FALSE;
            CraneLower := FALSE;
            IF CraneUp THEN
                _transit := TRUE;
                _state := Crane_states_t#Crane_Turn_Left_Metallic;
            END_IF;

        Crane_states_t#Crane_Lift_Magazine_White:
            _transit := FALSE;
            CraneLower := FALSE;
            IF CraneUp THEN
                _transit := TRUE;
                _state := Crane_states_t#Crane_Turn_Left_White;
            END_IF;

        Crane_states_t#Crane_Lift_NOT_Metallic_Black:
            _transit := FALSE;
            CraneLower := FALSE;
            IF CraneUp THEN
                _transit := TRUE;
                _state := Crane_states_t#Crane_Turn_Left_NOT_Metallic_Black;
            END_IF;

        Crane_states_t#Crane_Lower:
            _transit := FALSE;
            MagazinVacuumOn := TRUE;
            MagazinVacuumOff := FALSE;
            CraneLower := TRUE;
            AnalogCranePressure := INT#0;
            IF CraneSucked THEN
                _transit := TRUE;
                _state := Crane_states_t#Step0;
            END_IF;

        Crane_states_t#Crane_On_Conveyor:
            _transit := FALSE;
            CraneTurnCounterclockwise := FALSE;
            CraneTurnClockwise := FALSE;
            CraneLower := TRUE;
            IF CraneDown THEN
                _transit := TRUE;
                _state := Crane_states_t#release;
            END_IF;

        Crane_states_t#Crane_On_Conveyor_Metallic:
            _transit := FALSE;
            CraneTurnCounterclockwise := FALSE;
            CraneTurnClockwise := FALSE;
            CraneLower := TRUE;
            IF CraneDown THEN
                _transit := TRUE;
                _state := Crane_states_t#release;
            END_IF;

        Crane_states_t#Crane_On_Conveyor_Metallic2:
            _transit := FALSE;
            CraneTurnCounterclockwise := FALSE;
            CraneTurnClockwise := FALSE;
            CraneLower := TRUE;
            IF CraneDown THEN
                _transit := TRUE;
                _state := Crane_states_t#release2;
            END_IF;

        Crane_states_t#Crane_On_Conveyor_Not_Metallica_Black:
            _transit := FALSE;
            CraneTurnCounterclockwise := FALSE;
            CraneTurnClockwise := FALSE;
            CraneLower := TRUE;
            IF CraneDown THEN
                _transit := TRUE;
                _state := Crane_states_t#release_Black;
            END_IF;

        Crane_states_t#Crane_On_Stamp_Metallic:
            _transit := FALSE;
            CraneTurnCounterclockwise := FALSE;
            CraneTurnClockwise := FALSE;
            CraneLower := TRUE;
            IF CraneDown THEN
                _transit := TRUE;
                _state := Crane_states_t#release_Workpiece;
            END_IF;

        Crane_states_t#Crane_On_Stamp_Metallic2:
            _transit := FALSE;
            CraneTurnCounterclockwise := FALSE;
            CraneTurnClockwise := FALSE;
            IF StampLowered THEN
                _transit := TRUE;
                _state := Crane_states_t#Interstep_4;
            END_IF;

        Crane_states_t#Crane_On_Stamp_Metallic2_Lower:
            _transit := FALSE;
            CraneLower := TRUE;
            IF CraneDown THEN
                _transit := TRUE;
                _state := Crane_states_t#Suck_At_Stamp2;
            END_IF;

        Crane_states_t#Crane_On_Stamp_Stop_Black:
            _transit := FALSE;
            CraneTurnClockwise := FALSE;
            CraneTurnCounterclockwise := FALSE;
            IF TRUE THEN
                _transit := TRUE;
                _state := Crane_states_t#Reset_interconnect;
            END_IF;

        Crane_states_t#Crane_On_Stamp_White:
            _transit := FALSE;
            CraneTurnCounterclockwise := FALSE;
            CraneTurnClockwise := FALSE;
            CraneLower := TRUE;
            IF CraneDown THEN
                _transit := TRUE;
                _state := Crane_states_t#release_Workpiece_White;
            END_IF;

        Crane_states_t#Crane_Turn_Left_Back_To_Stamp:
            _transit := FALSE;
            CraneTurnCounterclockwise := TRUE;
            CraneTurnClockwise := FALSE;
            IF CranePositionStamp THEN
                _transit := TRUE;
                _state := Crane_states_t#Crane_On_Stamp_Stop_Black;
            END_IF;

        Crane_states_t#Crane_Turn_Left_From_Stamp:
            _transit := FALSE;
            CraneTurnClockwise := TRUE;
            CraneTurnCounterclockwise := FALSE;
            IF CraneOnConveyor THEN
                _transit := TRUE;
                _state := Crane_states_t#Crane_On_Conveyor_Metallic;
            END_IF;

        Crane_states_t#Crane_Turn_Left_Metallic:
            _transit := FALSE;
            CraneTurnCounterclockwise := TRUE;
            CraneTurnClockwise := FALSE;
            IF CranePositionStamp THEN
                _transit := TRUE;
                _state := Crane_states_t#Crane_On_Stamp_Metallic;
            END_IF;

        Crane_states_t#Crane_Turn_Left_Metallic2:
            _transit := FALSE;
            CraneTurnCounterclockwise := TRUE;
            CraneTurnClockwise := FALSE;
            IF CranePositionStamp THEN
                _transit := TRUE;
                _state := Crane_states_t#Crane_On_Stamp_Metallic2;
            END_IF;

        Crane_states_t#Crane_Turn_Left_NOT_Metallic:
            _transit := FALSE;
            CraneTurnCounterclockwise := TRUE;
            CraneTurnClockwise := FALSE;
            IF CraneOnConveyor THEN
                _transit := TRUE;
                _state := Crane_states_t#Crane_On_Conveyor;
            END_IF;

        Crane_states_t#Crane_Turn_Left_NOT_Metallic_Black:
            _transit := FALSE;
            CraneTurnCounterclockwise := TRUE;
            CraneTurnClockwise := FALSE;
            IF CraneOnConveyor THEN
                _transit := TRUE;
                _state := Crane_states_t#Crane_On_Conveyor_Not_Metallica_Black;
            END_IF;

        Crane_states_t#Crane_Turn_Left_White:
            _transit := FALSE;
            CraneTurnCounterclockwise := TRUE;
            CraneTurnClockwise := FALSE;
            IF CranePositionStamp THEN
                _transit := TRUE;
                _state := Crane_states_t#Crane_On_Stamp_White;
            END_IF;

        Crane_states_t#Crane_Turn_Right_From_Stamp:
            _transit := FALSE;
            CraneTurnClockwise := TRUE;
            CraneTurnCounterclockwise := FALSE;
            IF CraneOnConveyor THEN
                _transit := TRUE;
                _state := Crane_states_t#Crane_On_Conveyor_Metallic2;
            END_IF;

        Crane_states_t#Init:
            _transit := FALSE;
            IF TRUE THEN
                _transit := TRUE;
                _state := Crane_states_t#Start_Crane;
            END_IF;

        Crane_states_t#Interstep:
            _transit := FALSE;
            StartCommandCrane := TRUE;
            IF StartVar THEN
                _transit := TRUE;
                _state := Crane_states_t#Interstep_2;
            END_IF;

        Crane_states_t#Interstep_2:
            _transit := FALSE;
            IF SliderMovedOut THEN
                _transit := TRUE;
                _state := Crane_states_t#TimeDelay;
            END_IF;

        Crane_states_t#Interstep_3:
            _transit := FALSE;
            IF NOT WorkpieceReady THEN
                _transit := TRUE;
                _state := Crane_states_t#No_Workpiece_ready;
            ELSEIF WorkpieceReady THEN
                _transit := TRUE;
                _state := Crane_states_t#Turn_Right;
            END_IF;

        Crane_states_t#Interstep_4:
            _transit := FALSE;
            IF StampSliderSensorMovedOut THEN
                _transit := TRUE;
                _state := Crane_states_t#Crane_On_Stamp_Metallic2_Lower;
            END_IF;

        Crane_states_t#Lower_Crane:
            _transit := FALSE;
            CraneLower := TRUE;
            IF CraneDown THEN
                _transit := TRUE;
                _state := Crane_states_t#Suck_At_Stamp;
            END_IF;

        Crane_states_t#Magazin_Stop:
            _transit := FALSE;
            CraneTurnClockwise := FALSE;
            CraneTurnCounterclockwise := FALSE;
            IF TRUE THEN
                _transit := TRUE;
                _state := Crane_states_t#Crane_Lower;
            END_IF;

        Crane_states_t#Magazin_Stop_Black:
            _transit := FALSE;
            CraneTurnClockwise := FALSE;
            CraneTurnCounterclockwise := FALSE;
            MagazinVacuumOn := TRUE;
            MagazinVacuumOff := FALSE;
            CraneLower := TRUE;
            IF CraneSucked THEN
                _transit := TRUE;
                _state := Crane_states_t#Crane_Lift_NOT_Metallic_Black;
            END_IF;

        Crane_states_t#Magazin_Stop_Final:
            _transit := FALSE;
            CraneTurnClockwise := FALSE;
            CraneTurnCounterclockwise := FALSE;
            IF TRUE THEN
                _transit := TRUE;
                _state := Crane_states_t#Start_Crane;
            END_IF;

        Crane_states_t#No_Workpiece_ready:
            _transit := FALSE;
            MagazinVacuumOn := FALSE;
            MagazinVacuumOff := FALSE;
            CraneLower := FALSE;
            IF NOT StampSliderFilled THEN
                _transit := TRUE;
                _state := Crane_states_t#Turn_Right_Final;
            ELSEIF StampSliderFilled THEN
                _transit := TRUE;
                _state := Crane_states_t#Crane_Turn_Left_Metallic2;
            END_IF;

        Crane_states_t#Reset_interconnect:
            _transit := FALSE;
            interconnect := FALSE;
            Timer1(IN := FALSE, PT := TIME#1.0ms);
            IF SliderMovedOut THEN
                _transit := TRUE;
                _state := Crane_states_t#Lower_Crane;
            END_IF;

        Crane_states_t#Stamp_Pressure_Profile_Set_Metallic:
            _transit := FALSE;
            AnalogCranePressure := INT#7000;
            IF TRUE THEN
                _transit := TRUE;
                _state := Crane_states_t#Crane_Lift_Magazin_Metallic;
            END_IF;

        Crane_states_t#Stamp_Pressure_Profile_Set_White:
            _transit := FALSE;
            AnalogCranePressure := INT#6000;
            IF TRUE THEN
                _transit := TRUE;
                _state := Crane_states_t#Crane_Lift_Magazine_White;
            END_IF;

        Crane_states_t#Start_Crane:
            _transit := FALSE;
            CraneLower := FALSE;
            MagazinVacuumOff := TRUE;
            MagazinVacuumOn := FALSE;
            CraneTurnCounterclockwise := FALSE;
            CraneTurnClockwise := FALSE;
            StartVar := FALSE;
            StartCommandCrane := FALSE;
            IF (StartButtonMagazin = TRUE) THEN
                interconnectCraneStartCommand := TRUE;
            END_IF;
            IF interconnectCraneStartCommand THEN
                _transit := TRUE;
                _state := Crane_states_t#Crane_Init;
            END_IF;

        Crane_states_t#Step0:
            _transit := FALSE;
            IF (NOT MagazinCapacitiveSensor AND MagazinOpticalSensor) THEN
                _transit := TRUE;
                _state := Crane_states_t#Stamp_Pressure_Profile_Set_White;
            ELSEIF (MagazinCapacitiveSensor AND MagazinOpticalSensor) THEN
                _transit := TRUE;
                _state := Crane_states_t#Stamp_Pressure_Profile_Set_Metallic;
            ELSEIF (NOT MagazinCapacitiveSensor AND NOT MagazinOpticalSensor) THEN
                _transit := TRUE;
                _state := Crane_states_t#Crane_Lift_Magazin;
            END_IF;

        Crane_states_t#Step2:
            _transit := FALSE;
            IF (MagazinCapacitiveSensor OR MagazinOpticalSensor) THEN
                _transit := TRUE;
                _state := Crane_states_t#pause;
            ELSEIF (NOT MagazinCapacitiveSensor AND NOT MagazinOpticalSensor) THEN
                _transit := TRUE;
                _state := Crane_states_t#Turn_Right_Black;
            END_IF;

        Crane_states_t#Step3:
            _transit := FALSE;
            IF NOT WorkpieceReady THEN
                _transit := TRUE;
                _state := Crane_states_t#Step4;
            ELSEIF WorkpieceReady THEN
                _transit := TRUE;
                _state := Crane_states_t#Step2;
            END_IF;

        Crane_states_t#Step4:
            _transit := FALSE;
            IF TRUE THEN
                _transit := TRUE;
                _state := Crane_states_t#Interstep;
            END_IF;

        Crane_states_t#Suck_At_Stamp:
            _transit := FALSE;
            MagazinVacuumOn := TRUE;
            MagazinVacuumOff := FALSE;
            IF CraneSucked THEN
                _transit := TRUE;
                _state := Crane_states_t#Crane_Lift_At_Stamp;
            END_IF;

        Crane_states_t#Suck_At_Stamp2:
            _transit := FALSE;
            MagazinVacuumOn := TRUE;
            MagazinVacuumOff := FALSE;
            IF CraneSucked THEN
                _transit := TRUE;
                _state := Crane_states_t#Crane_Lift_At_Stamp2;
            END_IF;

        Crane_states_t#TimeDelay:
            _transit := FALSE;
            TimeDelay_Timer(IN := TRUE, PT := TimeDelay_Timer_Duration);
            TimeDelay_Timer_interconnect := TimeDelay_Timer.Q;
            IF TimeDelay_Timer_interconnect THEN
                _transit := TRUE;
                _state := Crane_states_t#Interstep_3;
            END_IF;

        Crane_states_t#Turn_Right:
            _transit := FALSE;
            CraneTurnClockwise := TRUE;
            CraneTurnCounterclockwise := FALSE;
            IF CraneOnMagazin THEN
                _transit := TRUE;
                _state := Crane_states_t#Magazin_Stop;
            END_IF;

        Crane_states_t#Turn_Right_Black:
            _transit := FALSE;
            CraneTurnClockwise := TRUE;
            CraneTurnCounterclockwise := FALSE;
            IF CraneOnMagazin THEN
                _transit := TRUE;
                _state := Crane_states_t#Magazin_Stop_Black;
            END_IF;

        Crane_states_t#Turn_Right_Final:
            _transit := FALSE;
            CraneTurnClockwise := TRUE;
            CraneTurnCounterclockwise := FALSE;
            AnalogCranePressure := INT#0;
            IF CraneOnMagazin THEN
                _transit := TRUE;
                _state := Crane_states_t#Magazin_Stop_Final;
            END_IF;

        Crane_states_t#pause:
            _transit := FALSE;
            Timer1(IN := CraneUp, PT := Duration1);
            interconnect := Timer1.Q;
            IF interconnect THEN
                _transit := TRUE;
                _state := Crane_states_t#Reset_interconnect;
            END_IF;

        Crane_states_t#release:
            _transit := FALSE;
            MagazinVacuumOff := TRUE;
            MagazinVacuumOn := FALSE;
            IF TRUE THEN
                _transit := TRUE;
                _state := Crane_states_t#Crane_Lift_Conveyor;
            END_IF;

        Crane_states_t#release2:
            _transit := FALSE;
            MagazinVacuumOff := TRUE;
            MagazinVacuumOn := FALSE;
            IF TRUE THEN
                _transit := TRUE;
                _state := Crane_states_t#Crane_Lift_Conveyor2;
            END_IF;

        Crane_states_t#release_Black:
            _transit := FALSE;
            MagazinVacuumOn := FALSE;
            MagazinVacuumOff := TRUE;
            IF TRUE THEN
                _transit := TRUE;
                _state := Crane_states_t#Crane_Lift_Conveyor_Black;
            END_IF;

        Crane_states_t#release_Workpiece:
            _transit := FALSE;
            MagazinVacuumOff := TRUE;
            MagazinVacuumOn := FALSE;
            IF TRUE THEN
                _transit := TRUE;
                _state := Crane_states_t#Crane_Go_Up;
            END_IF;

        Crane_states_t#release_Workpiece_White:
            _transit := FALSE;
            MagazinVacuumOff := TRUE;
            MagazinVacuumOn := FALSE;
            IF TRUE THEN
                _transit := TRUE;
                _state := Crane_states_t#Crane_Go_Up_White;
            END_IF;

            END_CASE;
END_FUNCTION_BLOCK

(* ---- Scenario8_Final.xml_Magazin.st ---- *)
FUNCTION_BLOCK Magazin
    VAR_INPUT  CraneDown : BOOL; END_VAR {*Irwxp*}
    VAR_OUTPUT  CraneLower : BOOL; END_VAR {*Orwxp*}
    VAR_INPUT  CraneOnConveyor : BOOL; END_VAR {*Irwxp*}
    VAR_INPUT  CraneOnMagazin : BOOL; END_VAR {*Irwxp*}
    VAR_INPUT  CraneSucked : BOOL; END_VAR {*Irwxp*}
    VAR_OUTPUT  CraneTurnClockwise : BOOL; END_VAR {*Orwxp*}
    VAR_OUTPUT  CraneTurnCounterclockwise : BOOL; END_VAR {*Orwxp*}
    VAR_INPUT  CraneUp : BOOL; END_VAR {*Irwxp*}
    VAR_OUTPUT  MagazinGreenLamp : BOOL; END_VAR {*Orwxp*}
    VAR_OUTPUT  MagazinSlider : BOOL; END_VAR {*Orwxp*}
    VAR_OUTPUT  MagazinVacuumOff : BOOL; END_VAR {*Orwxp*}
    VAR_OUTPUT  MagazinVacuumOn : BOOL; END_VAR {*Orwxp*}
    VAR_OUTPUT  MagazinWhiteLamp : BOOL; END_VAR {*Orwxp*}
    VAR  SFCInit : BOOL; END_VAR {*Lrwxp*}
    VAR_INPUT  SFCReset : BOOL; END_VAR {*Irwxp*}
    VAR_INPUT  SliderMovedOut : BOOL; END_VAR {*Irwxp*}
    VAR_INPUT  SliderNotMovedOut : BOOL; END_VAR {*Irwxp*}
    VAR_INPUT  StartButtonMagazin : BOOL; END_VAR {*Irwxp*}
    VAR_OUTPUT  StartCommandMagazin : BOOL; END_VAR {*Orwxp*}
    VAR_INPUT  StartVar : BOOL; END_VAR {*Irwxp*}
    VAR_INPUT  WorkpieceReady : BOOL; END_VAR {*Irwxp*}
    VAR  _state : Magazin_states_t; END_VAR {*Lrwxp*}
    VAR  _transit : BOOL; END_VAR {*Lrwxp*}
    VAR  interconnectMagazinStartCommand : BOOL; END_VAR {*Lrwxp*}

    CASE _state OF
        Magazin_states_t#Green_Lamp:
            _transit := FALSE;
            MagazinGreenLamp := TRUE;
            interconnectMagazinStartCommand := FALSE;
            IF TRUE THEN
                _transit := TRUE;
                _state := Magazin_states_t#Magazin_Init;
            END_IF;

        Magazin_states_t#Init:
            _transit := FALSE;
            IF TRUE THEN
                _transit := TRUE;
                _state := Magazin_states_t#Start_Magazin;
            END_IF;

        Magazin_states_t#Interstep:
            _transit := FALSE;
            StartCommandMagazin := TRUE;
            IF StartVar THEN
                _transit := TRUE;
                _state := Magazin_states_t#convey;
            END_IF;

        Magazin_states_t#Magazin_Init:
            _transit := FALSE;
            MagazinSlider := TRUE;
            IF TRUE THEN
                _transit := TRUE;
                _state := Magazin_states_t#Magazin_Init_2;
            END_IF;

        Magazin_states_t#Magazin_Init_2:
            _transit := FALSE;
            MagazinSlider := FALSE;
            IF TRUE THEN
                _transit := TRUE;
                _state := Magazin_states_t#Interstep;
            END_IF;

        Magazin_states_t#Slider_Move_Back:
            _transit := FALSE;
            IF ((SliderMovedOut = TRUE) AND (SliderNotMovedOut = FALSE)) THEN
                MagazinSlider := FALSE;
            END_IF;
            IF CraneUp THEN
                _transit := TRUE;
                _state := Magazin_states_t#Step1;
            END_IF;

        Magazin_states_t#Start_Magazin:
            _transit := FALSE;
            MagazinSlider := FALSE;
            MagazinGreenLamp := FALSE;
            StartVar := FALSE;
            StartCommandMagazin := FALSE;
            IF (StartButtonMagazin = TRUE) THEN
                interconnectMagazinStartCommand := TRUE;
            END_IF;
            IF interconnectMagazinStartCommand THEN
                _transit := TRUE;
                _state := Magazin_states_t#Green_Lamp;
            END_IF;

        Magazin_states_t#Step0:
            _transit := FALSE;
            IF CraneDown THEN
                _transit := TRUE;
                _state := Magazin_states_t#Slider_Move_Back;
            END_IF;

        Magazin_states_t#Step1:
            _transit := FALSE;
            IF CraneOnConveyor THEN
                _transit := TRUE;
                _state := Magazin_states_t#Interstep;
            END_IF;

        Magazin_states_t#convey:
            _transit := FALSE;
            IF SliderNotMovedOut THEN
                MagazinSlider := TRUE;
            END_IF;
            IF CraneOnMagazin THEN
                _transit := TRUE;
                _state := Magazin_states_t#Step0;
            END_IF;

            END_CASE;
END_FUNCTION_BLOCK

(* ---- Scenario8_Final.xml_Stamp.st ---- *)
FUNCTION_BLOCK Stamp
    VAR_INPUT  CraneDown : BOOL; END_VAR {*Irwxp*}
    VAR_INPUT  CraneOnConveyor : BOOL; END_VAR {*Irwxp*}
    VAR_INPUT  CranePositionStamp : BOOL; END_VAR {*Irwxp*}
    VAR_INPUT  CraneSucked : BOOL; END_VAR {*Irwxp*}
    VAR_INPUT  CraneUp : BOOL; END_VAR {*Irwxp*}
    VAR  Duration : TIME := TIME#500.0ms; END_VAR {*Lrwxp*}
    VAR  SFCInit : BOOL; END_VAR {*Lrwxp*}
    VAR_INPUT  SFCReset : BOOL; END_VAR {*Irwxp*}
    VAR_OUTPUT  StampGreenLamp : BOOL; END_VAR {*Orwxp*}
    VAR_INPUT  StampLowered : BOOL; END_VAR {*Irwxp*}
    VAR_OUTPUT  StampPressure : BOOL; END_VAR {*Orwxp*}
    VAR_OUTPUT  StampPusher : BOOL; END_VAR {*Orwxp*}
    VAR_INPUT  StampSliderFilled : BOOL; END_VAR {*Irwxp*}
    VAR_OUTPUT  StampSliderMovedIn : BOOL; END_VAR {*Orwxp*}
    VAR_OUTPUT  StampSliderMovedOut : BOOL; END_VAR {*Orwxp*}
    VAR_INPUT  StampSliderSensorMovedIn : BOOL; END_VAR {*Irwxp*}
    VAR_INPUT  StampSliderSensorMovedOut : BOOL; END_VAR {*Irwxp*}
    VAR_INPUT  StampStartButton : BOOL; END_VAR {*Irwxp*}
    VAR_INPUT  StampUp : BOOL; END_VAR {*Irwxp*}
    VAR_OUTPUT  StampWhiteLamp : BOOL; END_VAR {*Orwxp*}
    VAR_OUTPUT  StartCommandStamp : BOOL; END_VAR {*Orwxp*}
    VAR_INPUT  StartVar : BOOL; END_VAR {*Irwxp*}
    VAR  Timer : TON; END_VAR {*Lrwxp*}
    VAR  _state : Stamp_states_t; END_VAR {*Lrwxp*}
    VAR  _transit : BOOL; END_VAR {*Lrwxp*}
    VAR  interconnect : BOOL; END_VAR {*Lrwxp*}
    VAR  interconnectStampStartCommand : BOOL; END_VAR {*Lrwxp*}

    CASE _state OF
        Stamp_states_t#Green_Lamp:
            _transit := FALSE;
            StampGreenLamp := TRUE;
            interconnectStampStartCommand := FALSE;
            IF TRUE THEN
                _transit := TRUE;
                _state := Stamp_states_t#Stamp_Init_1;
            END_IF;

        Stamp_states_t#Init:
            _transit := FALSE;
            IF TRUE THEN
                _transit := TRUE;
                _state := Stamp_states_t#Start_Stamp;
            END_IF;

        Stamp_states_t#Interstep:
            _transit := FALSE;
            StartCommandStamp := TRUE;
            IF StartVar THEN
                _transit := TRUE;
                _state := Stamp_states_t#Interstep_2;
            END_IF;

        Stamp_states_t#Interstep_2:
            _transit := FALSE;
            IF StampSliderFilled THEN
                _transit := TRUE;
                _state := Stamp_states_t#Step0;
            END_IF;

        Stamp_states_t#StampProcess:
            _transit := FALSE;
            StampSliderMovedIn := FALSE;
            StampPusher := TRUE;
            IF StampLowered THEN
                _transit := TRUE;
                _state := Stamp_states_t#Step1;
            END_IF;

        Stamp_states_t#StampSliderBack:
            _transit := FALSE;
            StampSliderMovedIn := TRUE;
            StampSliderMovedOut := FALSE;
            IF StampSliderSensorMovedIn THEN
                _transit := TRUE;
                _state := Stamp_states_t#StampProcess;
            END_IF;

        Stamp_states_t#StampSliderForward:
            _transit := FALSE;
            StampPusher := FALSE;
            StampSliderMovedOut := TRUE;
            IF ((StampLowered = FALSE) AND (StampUp = TRUE)) THEN
                interconnect := FALSE;
            END_IF;
            Timer(IN := FALSE, PT := TIME#1.0ms);
            IF StampSliderMovedOut THEN
                _transit := TRUE;
                _state := Stamp_states_t#Step2;
            END_IF;

        Stamp_states_t#Stamp_Init_1:
            _transit := FALSE;
            StampSliderMovedIn := TRUE;
            StampSliderMovedOut := FALSE;
            IF StampSliderSensorMovedIn THEN
                _transit := TRUE;
                _state := Stamp_states_t#Stamp_Init_2;
            END_IF;

        Stamp_states_t#Stamp_Init_2:
            _transit := FALSE;
            StampSliderMovedIn := FALSE;
            StampSliderMovedOut := TRUE;
            IF StampSliderSensorMovedOut THEN
                _transit := TRUE;
                _state := Stamp_states_t#Stamp_Init_3;
            END_IF;

        Stamp_states_t#Stamp_Init_3:
            _transit := FALSE;
            StampPusher := TRUE;
            IF StampLowered THEN
                _transit := TRUE;
                _state := Stamp_states_t#Stamp_Init_4;
            END_IF;

        Stamp_states_t#Stamp_Init_4:
            _transit := FALSE;
            StampPusher := FALSE;
            IF StampUp THEN
                _transit := TRUE;
                _state := Stamp_states_t#Interstep;
            END_IF;

        Stamp_states_t#Start_Stamp:
            _transit := FALSE;
            StampSliderMovedOut := FALSE;
            StampSliderMovedIn := FALSE;
            StampPusher := FALSE;
            StampGreenLamp := FALSE;
            StampPressure := FALSE;
            StartCommandStamp := FALSE;
            IF (StampStartButton = TRUE) THEN
                interconnectStampStartCommand := TRUE;
            END_IF;
            IF interconnectStampStartCommand THEN
                _transit := TRUE;
                _state := Stamp_states_t#Green_Lamp;
            END_IF;

        Stamp_states_t#Step0:
            _transit := FALSE;
            IF CraneUp THEN
                _transit := TRUE;
                _state := Stamp_states_t#StampSliderBack;
            END_IF;

        Stamp_states_t#Step1:
            _transit := FALSE;
            Timer(IN := StampLowered, PT := TIME#);
            interconnect := Timer.Q;
            IF interconnect THEN
                _transit := TRUE;
                _state := Stamp_states_t#StampSliderForward;
            END_IF;

        Stamp_states_t#Step2:
            _transit := FALSE;
            IF (CraneOnConveyor AND NOT StampSliderFilled) THEN
                _transit := TRUE;
                _state := Stamp_states_t#Interstep;
            END_IF;

            END_CASE;
END_FUNCTION_BLOCK
